// TIA Portal V17 export
// export: Created 2025-03-05T08:02:25.9374573Z, ExportSetting WithDefaults, DisplayName Totally Integrated Automation Portal, DisplayVersion V17 Update 8, DisplayName TIA Portal Openness, DisplayVersion V17 Update 8, DisplayName TIA Portal Version Control Interface, DisplayVersion V17, DisplayName SINAMICS Startdrive Advanced, DisplayVersion V17 SP2, DisplayName SINAMICS Startdrive G110M, G120, G120C, G120D, G120P, G115D, DisplayVersion V17 SP2, DisplayName SINAMICS Startdrive G130, G150, S120, S150, SINAMICS MV, S210, DisplayVersion V17 SP2, DisplayName STEP 7 Professional, DisplayVersion V17 Update 8, DisplayName SINUMERIK ONE STEP 7 Toolbox, DisplayVersion V17 Update 12, DisplayName SINUMERIK 840D sl STEP 7 Toolbox, DisplayVersion V17 Update 12, DisplayName STEP 7 Safety, DisplayVersion V17 Update 6, DisplayName WinCC Advanced, DisplayVersion V17 Update 8
TYPE "CELL_SEQUENCES"
// stored: IsFailsafeCompliant false
   STRUCT
      GENERAL_CONDITIONS : Bool;   // GENERAL CONDITIONS
      INITIAL_CONDITIONS : Bool;   // INITIAL CONDITIONS
      START_REQUEST : Bool;   // START REQUEST
      START_COMMAND : Bool;   // START COMMAND
      SPARE_0_4 : Bool;   // SPARE 0 4
      COMMAND_PULSE : Bool;   // COMMAND PULSE
      REQUEST_PULSE : Bool;   // REQUEST PULSE
      SEQUENCE_RUNNING : Bool;   // SEQUENCE RUNNING
      STEP_1 : Bool;   // STEP 1
      STEP_2 : Bool;   // STEP 2
      STEP_3 : Bool;   // STEP 3
      STEP_4 : Bool;   // STEP 4
      STEP_5 : Bool;   // STEP 5
      STEP_6 : Bool;   // STEP 6
      STEP_7 : Bool;   // STEP 7
      STEP_8 : Bool;   // STEP 8
      STEP_9 : Bool;   // STEP 9
      STEP_10 : Bool;   // STEP 10
      STEP_11 : Bool;   // STEP 11
      STEP_12 : Bool;   // STEP 12
      STEP_13 : Bool;   // STEP 13
      STEP_14 : Bool;   // STEP 14
      STEP_15 : Bool;   // STEP 15
      STEP_16 : Bool;   // STEP 16
      SPARE_3_0 : Byte;   // SPARE 3 0
      SPARE_4_0 : Byte;   // SPARE 4 0
      RESET_PLC_CNC : Bool;   // RESET PLC CNC
      SEMI_REQ : Bool;   // SEMI REQUEST
      AUTO_REQ : Bool;   // AUTO REQUEST
      TEACH_PENDANT_REQUEST : Bool;   // TEACH PENDANT REQUEST
      SPARE_5_4 : Bool;   // SPARE 5 4
      SPARE_5_5 : Bool;   // SPARE 5 5
      SPARE_5_6 : Bool;   // SPARE 5 6
      SEQ_DONE : Bool;   // SEQ DONE
      TIME_EXCEEDED : Bool;   // TIME EXCEEDED
      SPARE_6_1 : Bool;   // SPARE 6 1
      SPARE_6_2 : Bool;   // SPARE 6 2
      SPARE_6_3 : Bool;   // SPARE 6 3
      SPARE_6_4 : Bool;   // SPARE 6 4
      SPARE_6_5 : Bool;   // SPARE 6 5
      SPARE_6_6 : Bool;   // SPARE 6 6
      SPARE_6_7 : Bool;   // SPARE 6 7
      WARNING : Bool;   // WARNING
      HELP : Bool;   // HELP
      SPARE_7_2 : Bool;   // SPARE 7 2
      SPARE_7_3 : Bool;   // SPARE 7 3
      SPARE_7_4 : Bool;   // SPARE 7 4
      SPARE_7_5 : Bool;   // SPARE 7 5
      SPARE_7_6 : Bool;   // SPARE 7 6
      SPARE_7_7 : Bool;   // SPARE 7 7
      AUX0 : Bool;   // AUX0
      AUX1 : Bool;   // AUX1
      AUX2 : Bool;   // AUX2
      AUX3 : Bool;   // AUX3
      WARNING_GONE : Bool;   // WARNING GONE
      AUX5 : Bool;   // AUX5
      AUX6 : Bool;   // AUX6
      AUX7 : Bool;   // AUX7
      START_GRAL_COND_HELP : Bool;   // START GENERAL COND HELP
      START_INIT_COND_HELP : Bool;   // START INITIAL COND HELP
      STOP_GRAL_HELP : Bool;   // STOP GENERAL HELP
      STOP_INIT_HELP : Bool;   // STOP INITIAL HELP
      SPARE_9_4 : Bool;   // SPARE 9 4
      SPARE_9_5 : Bool;   // SPARE 9 5
      GRAL_COND_HELP : Bool;   // GENERAL COND HELP
      INIT_COND_HELP : Bool;   // INITIAL COND HELP
      SPARE_10_0 : Byte;
      "TIMER_TIME _EXCEED" : TON_TIME;   // CELL SEQUENCE TIMER TIME EXCEEDED
   END_STRUCT;
   // "TIMER_TIME _EXCEED".PT := T#20S;
END_TYPE
